Staubli VAL3: OnF4.pgx

program OnF4()
  local num l_ni
begin
  //
  for l_ni=0 to 7
    sMsg[l_ni]=""
  endFor
  bPause=false
  //
  call Message("程序启动",true)

  //
  taskCreate "Mot",100,Motion()
  wait(taskStatus("Mot")==1)
  //信号
  taskCreate "sgd",100,takestop()
  wait(taskStatus("sgd")==1)
  //
  call Page()

end
